(* OutputValue := InputValue * (OutputMax - OutputMin)/(InputMax - InputMin) + OutputMin *)
FUNCTION_BLOCK AnalogScale
VAR_INPUT
	InputValue	: LREAL;
	InputMin	: LREAL:=0;
	InputMax	: LREAL:=100;
	OutputMin	: LREAL:=0;
	OutputMax	: LREAL:=100;
END_VAR
VAR_OUTPUT
	OutputValue	: LREAL;
	Percentage : LREAL;
	DataInvalid : BOOL;
END_VAR
VAR
END_VAR

IF InputMax - InputMin = 0 THEN
	DataInvalid := TRUE;
ELSE
	OutputValue := InputValue * (OutputMax - OutputMin)/(InputMax - InputMin) + OutputMin;
	Percentage := (InputValue - InputMin)/(InputMax - InputMin);
	DataInvalid := FALSE;
END_IF

END_FUNCTION_BLOCK

(* stored: Version 1.1.0.1, ProductVersion 3.1.4024.12
   POU AnalogScale: Id {515dce60-7141-4a80-87a8-389de0591337}, SpecialFunc None *)
